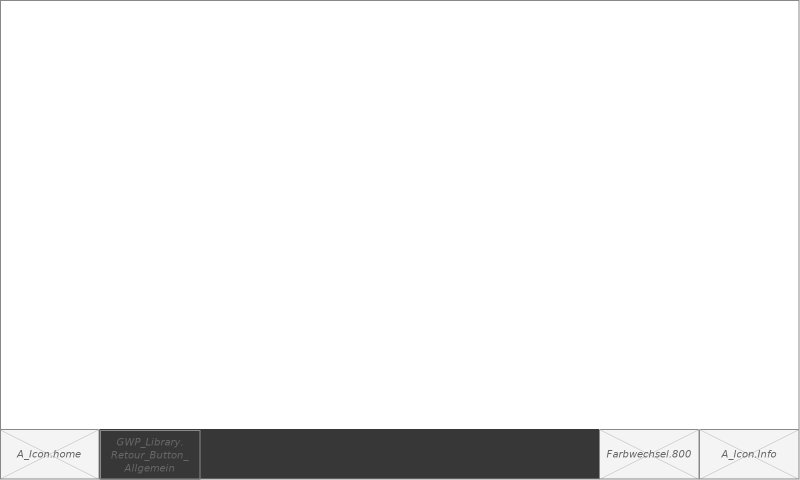
VISUALIZATION Fusszeile_50  // 800x480
    Rectangle (-1,429 800x50)
    Image (599,429 100x50), image: Farbwechsel.800
        p84334746: Visu.s_Status_AL_Button
        OnMouseClick: execute {
            visu.i_Frame_Index:=0;
            visu.i_Frame_KD_Index:=0;
            visu.i_Frame_KWP_Index:=0;
            visu.i_Frame_TWW_Index:=0;
            visu.i_Frame_VD_Index:=0;
            visu.i_Verschiebung_Horizontal:=0;
            visu.i_Verschiebung_Vertikal:=0;
            visu.i_Verschiebung_Vertikal_SW:=0;
            Alarmliste.Index:=0;
        }
        OnMouseClick: change screen: Alarmliste
    Image (699,429 100x50), image: A_Icon.Info
        OnMouseClick: execute {
            visu.i_Frame_Index:=0;
            visu.i_Frame_KD_Index:=0;
            visu.i_Frame_KWP_Index:=0;
            visu.i_Frame_TWW_Index:=0;
            visu.i_Frame_VD_Index:=0;
            visu.i_Verschiebung_Horizontal:=0;
            visu.i_Verschiebung_Vertikal:=0;
            visu.i_Verschiebung_Vertikal_SW:=0;
            Alarmliste.Index:=0;
        }
    Image (-1,429 100x50), image: A_Icon.home
        OnMouseClick: execute {
            visu.i_Frame_Index:=0;
            visu.i_Frame_KD_Index:=0;
            visu.i_Frame_KWP_Index:=0;
            visu.i_Frame_TWW_Index:=0;
            visu.i_Frame_VD_Index:=0;
            visu.i_Verschiebung_Horizontal:=0;
            visu.i_Verschiebung_Vertikal:=0;
            visu.i_Verschiebung_Vertikal_SW:=0;
            Alarmliste.Index:=0;
        }
        OnMouseClick: change screen: Home
    Frame (100,430 100x50)
        shows GWP_Library.Retour_Button_Allgemein()
END_VISUALIZATION

(* stored: Version 1.1.0.1, ProductVersion 3.1.4022.6
   Visu Fusszeile_50: Id {f05c05f2-fedb-467b-8f4d-bfd879d09530} *)
